TYPE ST_Ecat_State :
STRUCT
	wc_state : BOOL;
	op_state : UINT;
END_STRUCT
END_TYPE

(* stored: Version 1.1.0.1, ProductVersion 3.1.4024.12
   DUT ST_Ecat_State: Id {1aa4fd58-d47c-4bf6-a28c-8e29f3dd5b3c} *)
